VAR_GLOBAL
	G_sHMIAxisJogForward:				tsCoordinateBool;				//Axis jog forward
	G_sHMIAxisJogBackward:				tsCoordinateBool;				//Axis jog backward
END_VAR

(* stored: Version 1.1.0.1, ProductVersion 3.1.4022.18
   GVL HMI_GLV: Id {a928e4b6-8b64-4c92-bf20-994602f2ed71} *)
